// TIA Portal V17 export
// export: Created 2025-08-13T10:43:38.7127085Z, ExportSetting WithDefaults, DisplayName Totally Integrated Automation Portal, DisplayVersion V17 Update 8, DisplayName TIA Portal Openness, DisplayVersion V17 Update 8, DisplayName TIA Portal Version Control Interface, DisplayVersion V17, DisplayName SINAMICS Startdrive Advanced, DisplayVersion V17 SP2, DisplayName SINAMICS Startdrive G110M, G120, G120C, G120D, G120P, G115D, DisplayVersion V17 SP2, DisplayName SINAMICS Startdrive G130, G150, S120, S150, SINAMICS MV, S210, DisplayVersion V17 SP2, DisplayName STEP 7 Professional, DisplayVersion V17 Update 8, DisplayName STEP 7 Safety, DisplayVersion V17 Update 6, DisplayName WinCC Advanced, DisplayVersion V17 Update 8
ORGANIZATION_BLOCK "Main"   // OB1, LAD, ProgramCycle
TITLE = "Main Program Sweep (Cycle)"
{ S7_Optimized_Access := 'TRUE' }
VERSION : 0.1
// stored: AutoNumber true, IsIECCheckEnabled false, SetENOAutomatically false
   VAR_INPUT
      Initial_Call : Bool;   // Initial call of this OB
      Remanence : Bool;   // =True, if remanent data are available
   END_VAR
   VAR_TEMP
      Ack_Fault : Bool;
   END_VAR
BEGIN

REGION Network 1: Test Weld Sequence Reset
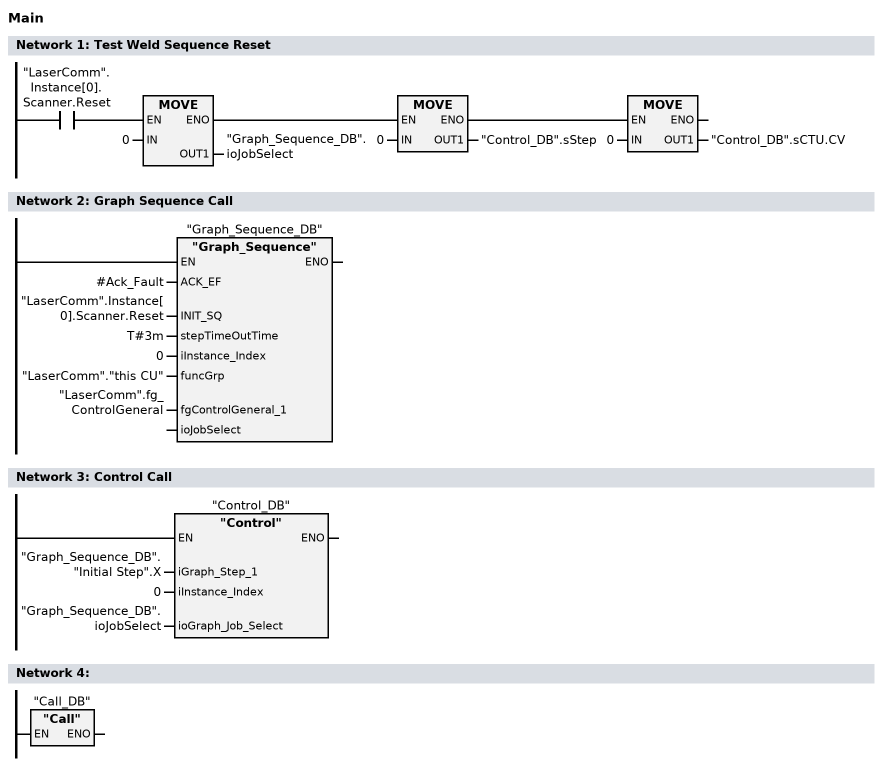
   RUNG wire#powerrail
      Contact( "LaserComm".Instance[0].Scanner.Reset )
      Move(in := 0, out1 => "Graph_Sequence_DB".ioJobSelect)
      Move(in := 0, out1 => "Control_DB".sStep)
      Move(in := 0, out1 => "Control_DB".sCTU.CV)
   END_RUNG
   // the same network as SCL:
   IF "LaserComm".Instance[0].Scanner.Reset THEN
       "Graph_Sequence_DB".ioJobSelect := 0;
       "Control_DB".sStep := 0;
       "Control_DB".sCTU.CV := 0;
   END_IF;
END_REGION

REGION Network 2: Graph Sequence Call
   RUNG wire#powerrail
      "Graph_Sequence_DB"(ACK_EF := #Ack_Fault, INIT_SQ := "LaserComm".Instance[0].Scanner.Reset, stepTimeOutTime := T#3m, iInstance_Index := 0, funcGrp := "LaserComm"."this CU", fgControlGeneral_1 := "LaserComm".fg_ControlGeneral, ioJobSelect :=)
   END_RUNG
   // the same network as SCL:
   "Graph_Sequence_DB"(ACK_EF := #Ack_Fault,   // "Graph_Sequence"
                       INIT_SQ := "LaserComm".Instance[0].Scanner.Reset,
                       stepTimeOutTime := T#3m,
                       iInstance_Index := 0,
                       funcGrp := "LaserComm"."this CU",
                       fgControlGeneral_1 := "LaserComm".fg_ControlGeneral);
END_REGION

REGION Network 3: Control Call
   RUNG wire#powerrail
      "Control_DB"(iGraph_Step_1 := "Graph_Sequence_DB"."Initial Step".X, iInstance_Index := 0, ioGraph_Job_Select := "Graph_Sequence_DB".ioJobSelect)
   END_RUNG
   // the same network as SCL:
   "Control_DB"(iGraph_Step_1 := "Graph_Sequence_DB"."Initial Step".X,   // "Control"
                iInstance_Index := 0,
                ioGraph_Job_Select := "Graph_Sequence_DB".ioJobSelect);
END_REGION

REGION Network 4
   RUNG wire#powerrail
      "Call_DB"()
   END_RUNG
   // the same network as SCL:
   "Call_DB"();   // "Call"
END_REGION
END_ORGANIZATION_BLOCK
